(* IEC 61131-3 sources: Std_PalletMover/Class/HAL_BMS_MasterVolt, 1 file *)

(* ---- HAL_BMS_MasterVolt.st ---- *)
#define HMI_ICON_CHARGING 12
#define LOWBATTERYCOMPARE 20
#define BATTERYCHARGINGDELAY 5 SEC

(*!
<Class
	Name               = "HAL_BMS_MasterVolt"
	Revision           = "0.0"
	RealtimeTask       = "false"
	CyclicTask         = "true"
	BackgroundTask     = "false"
	Sigmatek           = "false"
	OSInterface        = "false"
	HighPriority       = "false"
	Automatic          = "false"
	UpdateMode         = "Prescan"
	SharedCommandTable = "true"
	Objectsize         = "(840,900)">
	<Channels>
		<Server Name="BatteryAlarms" Visualized="false" Initialize="false" WriteProtected="true" Retentive="false"/>
		<Server Name="BatteryCharging" Visualized="false" Initialize="false" WriteProtected="true" Retentive="false"/>
		<Server Name="BatteryCurrent" Visualized="false" Initialize="false" WriteProtected="true" Retentive="false"/>
		<Server Name="BatteryTemperature" Visualized="false" Initialize="false" WriteProtected="true" Retentive="false"/>
		<Server Name="BatteryVirtualStateOfCharge" Visualized="true" Initialize="false" WriteProtected="true" Retentive="false"/>
		<Server Name="BatteryVoltage" Visualized="false" Initialize="false" WriteProtected="false" Retentive="false"/>
		<Server Name="EnergyDraw" Visualized="false" Initialize="false" WriteProtected="true" Retentive="false"/>
		<Server Name="HMIAdditionalIcon" Visualized="true" Initialize="false" WriteProtected="false" Retentive="false"/>
		<Server Name="HMIIconState" Visualized="true" Initialize="false" WriteProtected="false" Retentive="false"/>
		<Server Name="LowBatteryLimit" Visualized="false" Initialize="true" WriteProtected="false" Retentive="File"/>
		<Server Name="NMT" Visualized="false" Initialize="false" WriteProtected="true" Retentive="false"/>
		<Server Name="StateOfCharge" Visualized="false" Initialize="false" WriteProtected="false" Retentive="false"/>
		<Client Name="cNode" Required="true" Internal="false"/>
		<Client Name="Driver" Required="false" Internal="false"/>
		<Client Name="ObjCanOpenBase" Required="true" Internal="true"/>
	</Channels>
	<Separators>
		<Servers>
			<SepChn Position="10"/>
		</Servers>
	</Separators>
	<Network Name="HAL_BMS_MasterVolt">
		<!-- List of Components in this network -->
		<Components>
			<Object
				Name       = "_base"
				Class      = "HAL_BMS_Base"
				Position   = "(218,120)"
				Visualized = "false">
				<Channels>
					<Server Name="ClassSvr"/>
				</Channels>
			</Object>
			<Object
				Name       = "ObjCanOpenBase"
				Class      = "CanOpenWewoBase"
				Position   = "(210,420)"
				Visualized = "false"
				CyclicTime = "1 ms">
				<Channels>
					<Server Name="Server0"/>
					<Client Name="cNode"/>
					<Client Name="ConfigData"/>
					<Client Name="Driver"/>
				</Channels>
			</Object>
		</Components>
		<Comments>
		</Comments>
		<!-- List of Connections in this network -->
		<Connections>
			<Connection Source="this.ClassSvr" Destination="_base.ClassSvr" Vertices="(938,210),(518,210),"/>
			<Connection Source="this.ObjCanOpenBase" Destination="ObjCanOpenBase.Server0"/>
			<Connection Source="ObjCanOpenBase.Driver" Destination="this.Driver" Vertices="(210,510),(38,270),"/>
			<Connection Source="ObjCanOpenBase.cNode" Destination="this.cNode" Vertices="(210,570),(38,330),"/>
		</Connections>
		<!-- Headerfiles -->
		<Options>
		</Options>
	</Network>
</Class>
*)
#pragma using HAL_BMS_Base

HAL_BMS_MasterVolt : CLASS
: HAL_BMS_Base
	TYPE
	  tHMIAdditionalIconBMS :  //! <Type Public="true" Name="tHMIAdditionalIconBMS"/>
	  (
	    HAI_None,
	    HAI_Attention,
	    HAI_Charging
	  )$UDINT;
	END_TYPE
  //Servers:
	NMT 	: SvrCh_CanDeviceState_PTofCls_CanOpenBase;
	StateOfCharge 	: SvrCh_DINT;
	EnergyDraw 	: SvrCh_DINT;
	BatteryVoltage 	: SvrCh_DINT;
	BatteryCurrent 	: SvrCh_DINT;
	BatteryTemperature 	: SvrCh_DINT;
	BatteryAlarms 	: SvrCh_tBMSAlarms_PTofCls_HAL_BMS_Base;
	HMIIconState 	: SvrCh_DINT;
	HMIAdditionalIcon 	: SvrCh_tHMIAdditionalIconBMS_PTofCls_HAL_BMS_MasterVolt;
	BatteryCharging 	: SvrCh_DINT;
	LowBatteryLimit 	: SvrCh_DINT;
	BatteryVirtualStateOfCharge 	: SvrCh_DINT;
  //Clients:
	Driver 	: CltChCmd_CanDriverBase;
	cNode 	: CltCh_DINT;
	ObjCanOpenBase 	: CltChCmd_CanOpenWewoBase;
  //Variables:
		_pdoIn1 	: PDOStr;
		_pdoIn2 	: PDOStr;
		_pdoIn3 	: PDOStr;
		_pdoIn4 	: PDOStr;
		_pdo1rxTime 	: UDINT;
		_pdo2rxTime 	: UDINT;
		_pdo3rxTime 	: UDINT;
		_pdo4rxTime 	: UDINT;
		_pdo1RxInterval 	: UDINT;
		_pdo2RxInterval 	: UDINT;
		_pdo3RxInterval 	: UDINT;
		_startUpDelayPassed 	: BOOL;
		_initCounter 	: DINT;
		_batteryChargingTimer 	: UDINT;
  //Functions:

	FUNCTION VIRTUAL GLOBAL Init;

	FUNCTION VIRTUAL GLOBAL CyWork
		VAR_INPUT
			EAX 	: UDINT;
		END_VAR
		VAR_OUTPUT
			state (EAX) 	: UDINT := READY;
		END_VAR;

	FUNCTION VIRTUAL GLOBAL GetBMSData
		VAR_OUTPUT
			returnValue 	: tBMSData;
		END_VAR;

	FUNCTION _receiveData;

	FUNCTION _handleAlarms;

	FUNCTION _handleAlarmResets;
  //Tables:
	FUNCTION @STD
		VAR_OUTPUT
			ret_code	: CONFSTATES;
		END_VAR;
	FUNCTION GLOBAL TAB @CT_;
END_CLASS;

#pragma using CanOpenWewoBase
#pragma usingLtd CanDriverBase

FUNCTION VIRTUAL GLOBAL HAL_BMS_MasterVolt::Init
  _initCounter += 1;

 END_FUNCTION

FUNCTION VIRTUAL GLOBAL HAL_BMS_MasterVolt::CyWork
	VAR_INPUT
		EAX 	: UDINT;
	END_VAR
	VAR_OUTPUT
		state (EAX) 	: UDINT;(* := READY *)
	END_VAR

  _receiveData();

  if ops.tAbsolute > TIMEOUTDELAY then
    _startUpDelayPassed := TRUE;
  end_if;

  if  (_startUpDelayPassed = TRUE) & ( (ops.tAbsolute - _pdo1rxTime) > COMM_TIMEOUT | (ops.tAbsolute - _pdo2rxTime) > COMM_TIMEOUT | (ops.tAbsolute - _pdo3rxTime) > COMM_TIMEOUT ) then
    // Activate timeout alarm if the cyclic messages aren't received or sent in time.
    BatteryAlarms.ba_NoCommunication := TRUE;
  else
    BatteryAlarms.ba_NoCommunication := FALSE;
  end_if;

  BatteryVirtualStateOfCharge := 100*(StateOfCharge - LowBatteryLimit)/(100 - LowBatteryLimit);
  HMIIconState := BatteryVirtualStateOfCharge/20;
  BatteryCharging := (BatteryCurrent > 0);

  if BatteryCharging = TRUE then
    HMIIconState := HMI_ICON_CHARGING;
  end_if;

END_FUNCTION

FUNCTION VIRTUAL GLOBAL HAL_BMS_MasterVolt::GetBMSData
	VAR_OUTPUT
		returnValue 	: tBMSData;
	END_VAR

  returnValue.bd_StateOfCharge := to_uint(StateOfCharge);
  // returnValue.bd_TimeToGo :=
  returnValue.bd_EnergyDraw := to_int(EnergyDraw);
  returnValue.bd_BatteryVoltage := to_uint(BatteryVoltage);
  returnValue.bd_BatteryCurrent := to_int(BatteryCurrent);
  returnValue.bd_BatteryTemperature := to_int(BatteryTemperature);
  returnValue.bd_BatteryCharging := to_bool(BatteryCharging);
  returnValue.bd_BatteryLowIndication := (BatteryVirtualStateOfCharge <= LOWBATTERYCOMPARE);
  returnValue.bd_Alarm := BatteryAlarms;

END_FUNCTION

FUNCTION HAL_BMS_MasterVolt::_receiveData
  VAR
  	tmpDataReceived : BOOL;
    tmpBMSData      : tBMSData;
  END_VAR

  tmpDataReceived := FALSE;

  //----------------------------------------------------
  // Read out PDO_RX1 with identifier 0x180 + NodeID
  //----------------------------------------------------
  if ObjCanOpenBase.DecoPDO(PdoId:= cPdoRx1, Value1:= #_pdoIn1.Val1, Value2:= #_pdoIn1.Val2, Value3:= #_pdoIn1.Val3, Value4:= #_pdoIn1.Val4) = 0 then
    // Received value
    _pdo1RxInterval := (ops.tAbsolute - _pdo1rxTime);
    _pdo1rxTime := ops.tAbsolute;    // time the valid response was receive

    StateOfCharge := to_dint(_pdoIn1.Val1);
    EnergyDraw := to_dint(_pdoIn1.Val2);
    BatteryVoltage := to_dint(_pdoIn1.Val3);
    BatteryCurrent := to_dint(_pdoIn1.Val4);
    tmpDataReceived := TRUE;

  end_if;

  //----------------------------------------------------
  // Read out PDO_RX2 with identifier 0x280 + NodeID
  //----------------------------------------------------
  if ObjCanOpenBase.DecoPDO(PdoId:= cPdoRx2, Value1:= #_pdoIn2.Val1, Value2:= #_pdoIn2.Val2, Value3:= #_pdoIn2.Val3, Value4:= #_pdoIn2.Val4) = 0 then
    // Received value
    _pdo2RxInterval := (ops.tAbsolute - _pdo2rxTime);
    _pdo2rxTime := ops.tAbsolute;    // time the valid response was receive

    BatteryTemperature := to_dint(_pdoIn2.Val1);
    BatteryAlarms.ba_OverVoltage := _pdoIn2.Val2$BOOL;
    BatteryAlarms.ba_UnderVoltage := _pdoIn2.Val3$BOOL;
    BatteryAlarms.ba_BatteryEmpty := _pdoIn2.Val4$BOOL;
    tmpDataReceived := TRUE;

  end_if;

  //----------------------------------------------------
  // Read out PDO_RX3 with identifier 0x380 + NodeID
  //----------------------------------------------------
  if ObjCanOpenBase.DecoPDO(PdoId:= cPdoRx3, Value1:= #_pdoIn3.Val1, Value2:= #_pdoIn3.Val2, Value3:= #_pdoIn3.Val3, Value4:= #_pdoIn3.Val4) = 0 then
    // Received value
    _pdo3RxInterval := (ops.tAbsolute - _pdo3rxTime);
    _pdo3rxTime := ops.tAbsolute;    // time the valid response was receive

    BatteryAlarms.ba_InternalDefect := _pdoIn3.Val1$BOOL;
    BatteryAlarms.ba_AlmostUnderVoltage := _pdoIn3.Val2$BOOL;
    BatteryAlarms.ba_BatteryAlmostEmpty := _pdoIn3.Val3$BOOL;
    tmpDataReceived := TRUE;

  end_if;

 // If NMT state is not operational, send it to operational
  if ObjCanOpenBase.DecoNMT(NmtId:=cNmtErr, DeviceState:=#NMT) = 0 then
    if NMT <> CanOpenBase::cds_Operational then
      ObjCanOpenBase.BuildNmt(NmtId:=0, Cmnd:=1, Node:=cNode);
    end_if;
  end_if;

  if tmpDataReceived = TRUE then

    tmpBMSData.bd_StateOfCharge := to_uint(BatteryVirtualStateOfCharge);
    //tmpBMSData.bd_TimeToGo :=
    tmpBMSData.bd_EnergyDraw := to_int(EnergyDraw);
    tmpBMSData.bd_BatteryVoltage := to_uint(BatteryVoltage);
    tmpBMSData.bd_BatteryCurrent := to_int(BatteryCurrent);
    tmpBMSData.bd_BatteryTemperature := to_int(BatteryTemperature);

    if BatteryCurrent <= 0 then
      _batteryChargingTimer := ops.tAbsolute;
    end_if;

    tmpBMSData.bd_BatteryCharging := ((ops.tAbsolute - _batteryChargingTimer) > BATTERYCHARGINGDELAY);
    tmpBMSData.bd_Alarm := BatteryAlarms;

  end_if;

END_FUNCTION

FUNCTION HAL_BMS_MasterVolt::_handleAlarms

  if BatteryAlarms.ba_OverVoltage = TRUE then

  end_if;

  if BatteryAlarms.ba_UnderVoltage = TRUE then

  end_if;

  if BatteryAlarms.ba_AlmostUnderVoltage = TRUE then

  end_if;

  if BatteryAlarms.ba_BatteryEmpty = TRUE then

  end_if;

  if BatteryAlarms.ba_BatteryAlmostEmpty = TRUE then

  end_if;

  if BatteryAlarms.ba_InternalDefect = TRUE then

  end_if;

  if BatteryAlarms.ba_NoCommunication = TRUE then

  end_if;

END_FUNCTION

FUNCTION HAL_BMS_MasterVolt::_handleAlarmResets

END_FUNCTION
